{attribute 'qualified_only'}
VAR_GLOBAL
	myVeryFirstDatamanGVL 	: TcoCognexVision.TcoDatamanIO_v_5_x_x;
END_VAR

(* stored: Version 1.1.0.1, ProductVersion 3.1.4024.11
   GVL GVL: Id {f49b796b-e857-0a7c-1c6a-0b51ef76ee8b} *)
